{attribute 'qualified_only'}
{attribute 'strict'}
{attribute 'to_string'}
TYPE E_Severity :
(
	Alarm := 1,
	Warning
);
END_TYPE

(* stored: Version 1.1.0.1, ProductVersion 3.1.4026.18
   DUT E_Severity: Id {78eb8743-b0f2-4e7a-befc-576684a31bf8} *)
